INTERFACE ITF_BaseComponent

END_INTERFACE

(* stored: Version 1.1.0.1
   Itf ITF_BaseComponent: Id {bfd259ad-b5a7-0c3e-25af-f416d786cc1f} *)
